FUNCTION_BLOCK CAT1 (* Composite Function Block Type *)
  (* Standard: 61499-2 *)
  (* Version 0.0, 12/04/2022, labor, Schneider Electric, template *)
  PACKAGE Main;
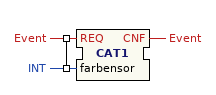
  EVENT_INPUT
    REQ WITH farbensor; (* Normal Execution Request *)
  END_EVENT
  EVENT_OUTPUT
    CNF; (* Execution Confirmation *)
  END_EVENT
  VAR_INPUT
    farbensor : INT;
  END_VAR
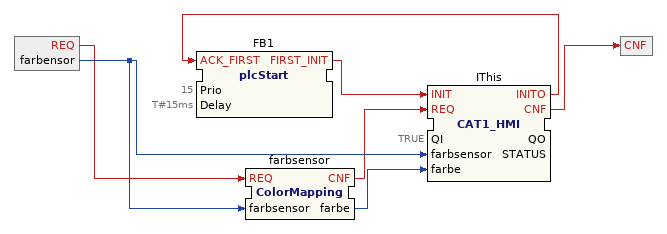
  FBS
    IThis : CAT1_HMI(QI := TRUE);
    FB1 : plcStart(Prio := 15, Delay := T#15ms);
    farbsensor : ColorMapping;
  END_FBS
  EVENT_CONNECTIONS
    REQ TO farbsensor.REQ;
    FB1.FIRST_INIT TO IThis.INIT;
    farbsensor.CNF TO IThis.REQ;
    IThis.INITO TO FB1.ACK_FIRST;
    IThis.CNF TO CNF;
  END_CONNECTIONS
  DATA_CONNECTIONS
    farbensor TO farbsensor.farbsensor;
    farbensor TO IThis.farbsensor;
    farbsensor.farbe TO IThis.farbe;
  END_CONNECTIONS
END_FUNCTION_BLOCK
